INTERFACE I_Tag EXTENDS Debug.I_Debug

PROPERTY Cache : UDINT
GET
END_GET
END_PROPERTY

METHOD GetId : Strings.Str
VAR_INPUT
END_VAR
END_METHOD

METHOD Join : Results.Result
VAR_INPUT
	iOwner		: I_TagOwner;
	nCache		: UDINT;
END_VAR
END_METHOD

METHOD Leave : Results.Result
VAR_INPUT
	iOwner		: I_TagOwner;
END_VAR
END_METHOD

PROPERTY Option : Strings.Str
GET
END_GET
END_PROPERTY

PROPERTY Owner : I_TagOwner
GET
END_GET
END_PROPERTY

PROPERTY Self : I_Tag
GET
END_GET
END_PROPERTY

END_INTERFACE

(* stored: Version 1.1.0.1
   Itf I_Tag: Id {169b0aa9-3f7f-4d5f-86c3-0a839d1aeed2}
   Property Cache: Id {a7a9550e-d99f-4348-a33b-ef0f866499c2}
   Get Get: Id {6c2e3446-d7b5-413d-95eb-b107e3803b1e}
   Method GetId: Id {a672ec3d-a76e-46ac-b519-eab39d5b74fc}
   Method Join: Id {eb215011-c9cf-4297-98dd-50dbfcfe4dab}
   Method Leave: Id {ed0ad921-8e92-48f7-a6d2-3d783d92be69}
   Property Option: Id {6cb9ccec-1ce6-4897-90e2-ce07ec9d308b}
   Get Get: Id {85cb6215-8cbc-4e1d-8f0e-c96079b830e7}
   Property Owner: Id {c3357166-aa2c-47c6-b394-c75ee3f8942e}
   Get Get: Id {8f4fa24a-1004-42f9-b338-5ebee0680709}
   Property Self: Id {31adaab0-78c5-4e17-9514-7846bfb1d186}
   Get Get: Id {cbe7d038-f895-4e3c-bffa-766279a6771c} *)
